% RSLogix 500 project PID_Logic_Vaccum.RSS, saved by version 8.30.00.16 %
PROJECT "UNTITLED"    % processor: Bul.1763 MicroLogix 1100 Series B %

PROGRAM FILES
  LAD 2   4 rungs
  LAD 3 "IO"  3 rungs
  LAD 4 "CTRL"  11 rungs

DATA FILES
  O0 OUTPUT  4 elements
  I1 INPUT  6 elements
  S2 STATUS  66 elements
  B3 BINARY  1 elements
  T4 TIMER  1 elements
  C5 COUNTER  1 elements
  R6 CONTROL  1 elements
  N7 INTEGER  7 elements
  F8 FLOAT  2 elements

LADDER 2
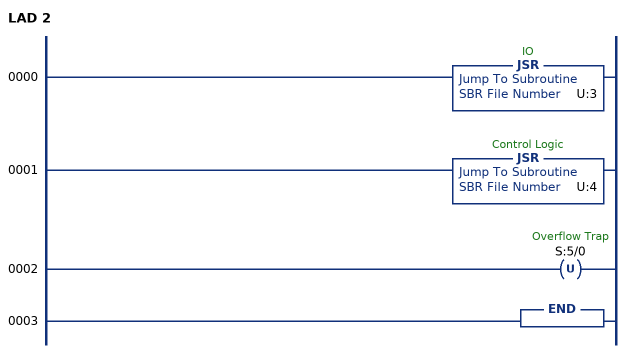
% Rung: 0 %
SOR JSR U:3 EOR
%   U:3  "IO" %
% Rung: 1 %
SOR JSR U:4 EOR
%   U:4  "Control Logic" %
% Rung: 2 %
SOR OTU S:5/0 EOR
%   S:5/0  "Overflow Trap" %
% Rung: 3 %
SOR END EOR

LADDER 3 "IO"
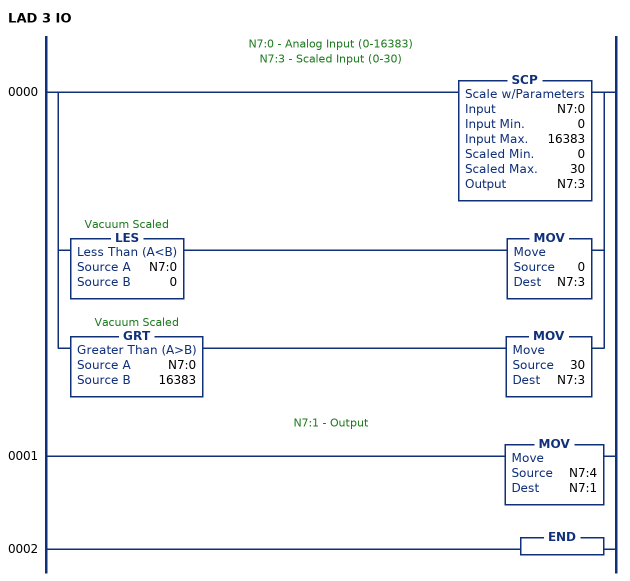
% Rung: 0 %
% N7:0 - Analog Input (0-16383)
% N7:3 - Scaled Input (0-30) %
SOR BST BST SCP N7:0 0 16383 0 30 N7:3 NXB LES N7:0 0 MOV 0 N7:3 BND NXB GRT N7:0 16383 MOV 30 N7:3 BND EOR
%   N7:0  "Vacuum Scaled" %
% Rung: 1 %
% N7:1 - Output %
SOR MOV N7:4 N7:1 EOR
% Rung: 2 %
SOR END EOR

LADDER 4 "CTRL"
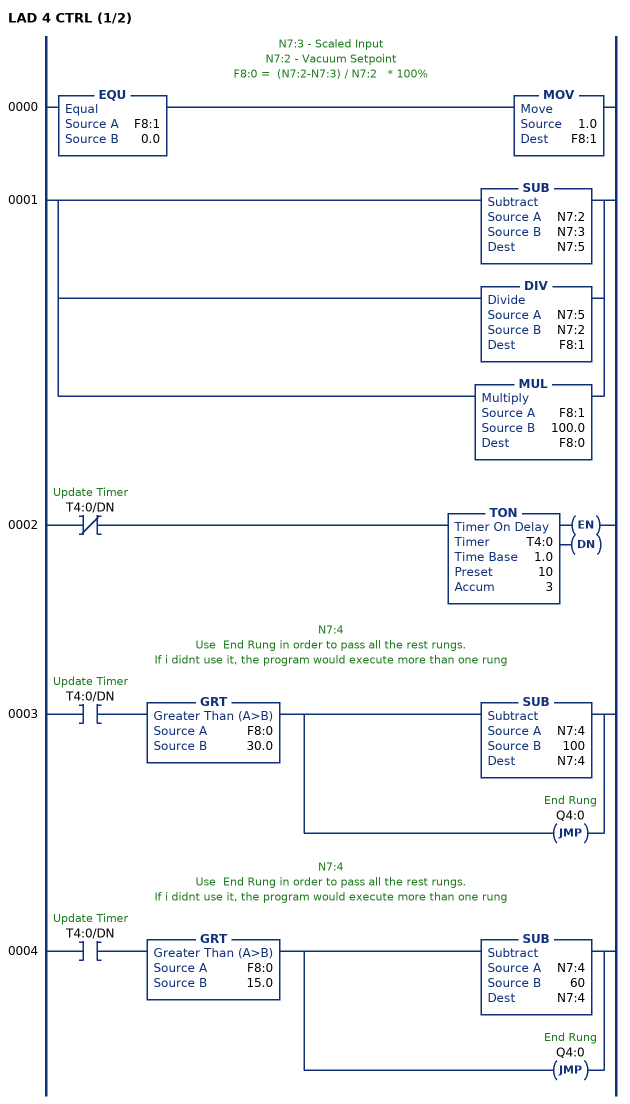
% Rung: 0 %
% N7:3 - Scaled Input
% N7:2 - Vacuum Setpoint
% 
% F8:0 =  (N7:2-N7:3) / N7:2   * 100% %
SOR EQU F8:1 0.0 MOV 1.0 F8:1 EOR
% Rung: 1 %
SOR BST BST SUB N7:2 N7:3 N7:5 NXB DIV N7:5 N7:2 F8:1 BND NXB MUL F8:1 100.0 F8:0 BND EOR
%   N7:2  "Vacuum Setpoint" %
% Rung: 2 %
SOR XIO T4:0/DN TON T4:0 1.0 10 3 EOR
%   T4:0/DN  "Update Timer" %
% Rung: 3 %
% N7:4
% 
% Use  End Rung in order to pass all the rest rungs.
% If i didnt use it, the program would execute more than one rung %
SOR XIC T4:0/DN GRT F8:0 30.0 BST SUB N7:4 100 N7:4 NXB JMP Q4:0 BND EOR
%   T4:0/DN  "Update Timer" %
%   Q4:0  "End Rung" %
% Rung: 4 %
% N7:4
% 
% Use  End Rung in order to pass all the rest rungs.
% If i didnt use it, the program would execute more than one rung %
SOR XIC T4:0/DN GRT F8:0 15.0 BST SUB N7:4 60 N7:4 NXB JMP Q4:0 BND EOR
%   T4:0/DN  "Update Timer" %
%   Q4:0  "End Rung" %

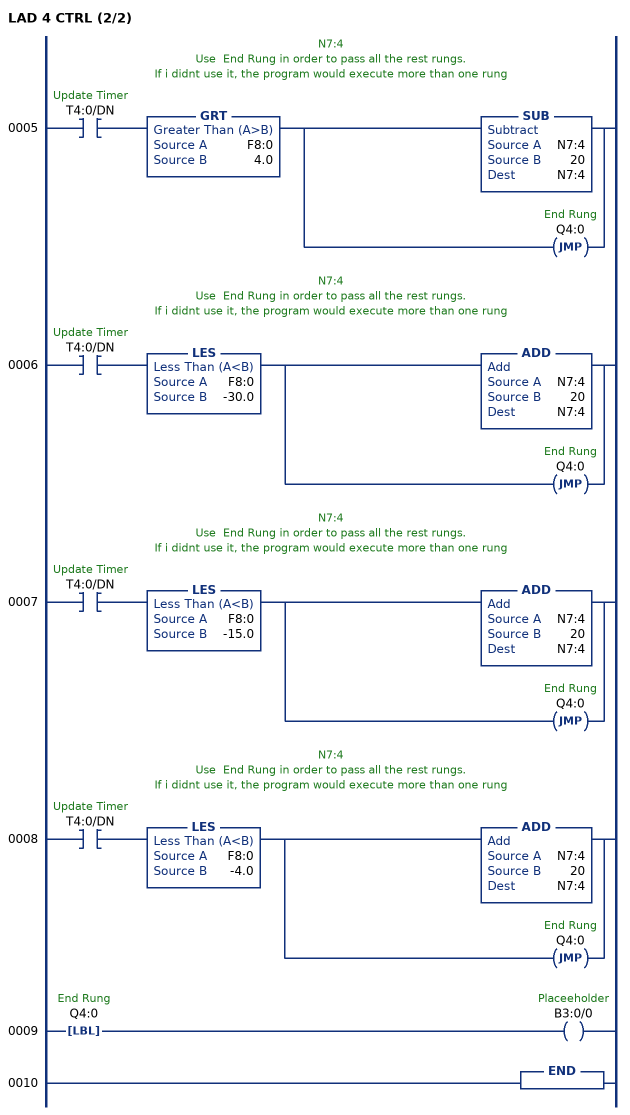
% Rung: 5 %
% N7:4
% 
% Use  End Rung in order to pass all the rest rungs.
% If i didnt use it, the program would execute more than one rung %
SOR XIC T4:0/DN GRT F8:0 4.0 BST SUB N7:4 20 N7:4 NXB JMP Q4:0 BND EOR
%   T4:0/DN  "Update Timer" %
%   Q4:0  "End Rung" %
% Rung: 6 %
% N7:4
% 
% Use  End Rung in order to pass all the rest rungs.
% If i didnt use it, the program would execute more than one rung %
SOR XIC T4:0/DN LES F8:0 -30.0 BST ADD N7:4 20 N7:4 NXB JMP Q4:0 BND EOR
%   T4:0/DN  "Update Timer" %
%   Q4:0  "End Rung" %
% Rung: 7 %
% N7:4
% 
% Use  End Rung in order to pass all the rest rungs.
% If i didnt use it, the program would execute more than one rung %
SOR XIC T4:0/DN LES F8:0 -15.0 BST ADD N7:4 20 N7:4 NXB JMP Q4:0 BND EOR
%   T4:0/DN  "Update Timer" %
%   Q4:0  "End Rung" %
% Rung: 8 %
% N7:4
% 
% Use  End Rung in order to pass all the rest rungs.
% If i didnt use it, the program would execute more than one rung %
SOR XIC T4:0/DN LES F8:0 -4.0 BST ADD N7:4 20 N7:4 NXB JMP Q4:0 BND EOR
%   T4:0/DN  "Update Timer" %
%   Q4:0  "End Rung" %
% Rung: 9 %
SOR LBL Q4:0 OTE B3:0/0 EOR
%   Q4:0  "End Rung" %
%   B3:0/0  "Placeeholder" %
% Rung: 10 %
SOR END EOR

DATA TABLE (non-zero values as saved)
DATA B3
% B3:0 % 0X0001
DATA T4
% .PRE .ACC %
% T4:0 % 10 3
DATA N7
% N7:0 % 8750 4700 15 16 0 -1 0
DATA F8
% F8:0 % -6.666667 -0.06666667
